// TIA Portal project "Analog Raw" (V17)

(* hardware
DEVICE "S7-1200 station_1"  S7-1200 Station
   slot 0: "Rack_0"  S7-1200 Rack  Rack  V1.0
   slot 1: "PLC_1"  CPU 1217C DC/DC/DC  6ES7 217-1AG40-0XB0  V4.5
   slot 2: "AI 4x13BIT_1"  6ES7 231-4HD32-0XB0  V2.1
*)

// ===== PLC "PLC_1"  CPU 1217C DC/DC/DC =====

VAR_GLOBAL   // PLC tag table "Default tag table"
   "Raw_Level" AT %MW10 : Int;
   "Normalized_Level" AT %MD20 : Real;
   "Tank_Level_Percent" AT %MD24 : Real;
END_VAR

ORGANIZATION_BLOCK "Main"   // OB1, LAD, ProgramCycle
TITLE = "Main Program Sweep (Cycle)"
{ S7_Optimized_Access := 'TRUE' }
VERSION : 0.1
   VAR_INPUT
      Initial_Call : Bool;   // Initial call of this OB
      Remanence : Bool;   // =True, if remanent data are available
   END_VAR
BEGIN

REGION Network 1
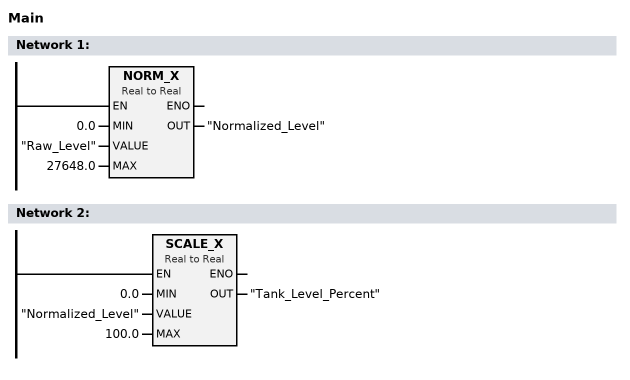
   RUNG wire#powerrail
      { S7_Templates := "[SrcType := Real, DestType := Real]" } Normalize(min := 0.0, value := "Raw_Level", max := 27648.0, out => "Normalized_Level")
   END_RUNG
   // the same network as SCL:
   "Normalized_Level" := NORM_X(MIN := 0.0, VALUE := "Raw_Level", MAX := 27648.0);
END_REGION

REGION Network 2
   RUNG wire#powerrail
      { S7_Templates := "[SrcType := Real, DestType := Real]" } Scale(min := 0.0, value := "Normalized_Level", max := 100.0, out => "Tank_Level_Percent")
   END_RUNG
   // the same network as SCL:
   "Tank_Level_Percent" := SCALE_X(MIN := 0.0, VALUE := "Normalized_Level", MAX := 100.0);
END_REGION
END_ORGANIZATION_BLOCK